{attribute 'qualified_only'}
{attribute 'strict'}
TYPE StateActuator :
(
	None,
	Error,
	Retracting,
	Retracted,
	Extending,
	Extended
);
END_TYPE

(* stored: Version 1.1.0.1, ProductVersion 3.1.4022.11
   DUT StateActuator: Id {054d0146-6ed0-4540-a536-553e6061ddbd} *)
